// TIA Portal project "2022.06.13_步进电机定位指令" (V17)

(* hardware
DEVICE "S7-1200 station_1"  S7-1200 Station
   slot 0: "Rack_0"  S7-1200 Rack  Rack  V1.0
   slot 1: "PLC_1"  CPU 1212C DC/DC/DC  6ES7 212-1AE40-0XB0  V4.5
   slot 2: "AI 4x13BIT/AQ 2x14BIT_1"  SM 1234 AI4/AQ2  6ES7 234-4HE30-0XB0  V1.0
*)

// ===== PLC "PLC_1"  CPU 1212C DC/DC/DC =====

VAR_GLOBAL   // PLC tag table "默认变量表"
   "液位测量" AT %IW96 : Word;
   "百分比" AT %MD40 : DWord;
   "模拟量输出通道" AT %MD44 : UDInt;
   "所需频率(1)" AT %MD0 : Real;
   "压力2模拟输入通道" AT %IW100 : Int;
   "液位" AT %MD4 : Real;
   "频率" AT %MD8 : Real;
   "Tag_2" AT %MD12 : Real;
   "模拟量输出" AT %QW96 : Int;
   "设定液位值" AT %MD20 : Real;
   "实际液位值" AT %MD24 : Real;
   "轴_1_脉冲" AT %Q0.0 : Bool;
   "轴_1_方向" AT %Q0.1 : Bool;
   "轴_1_LowHwLimitSwitch" AT %I0.0 : Bool;
   "轴_1_HighHwLimitSwitch" AT %I0.1 : Bool;
   "轴_1_PassiveHomingSwitch" AT %I0.2 : Bool;
   "轴_1_归位开关" AT %I0.3 : Bool;
   "启用轴" AT %M0.0 : Bool;
   "完成位" AT %M0.1 : Bool;
   "Tag_1" AT %M0.2 : Bool;
   "回原点" AT %I1.0 : Bool;
   "Tag_3" AT %M0.4 : Bool;
   "Tag_4" AT %M0.5 : Bool;
   "Tag_5" AT %M0.3 : Bool;
   "触发绝对定位" AT %I1.1 : Bool;
   "Tag_7" AT %M0.6 : Bool;
   "指定位置" AT %MD30 : Real;
   "指定速度" AT %MD34 : Real;
   "Tag_6" AT %M0.7 : Bool;
   "Tag_8" AT %I1.2 : Bool;
   "Tag_9" AT %M1.0 : Bool;
   "触发相对位移指令" AT %I1.3 : Bool;
   "Tag_11" AT %M1.1 : Bool;
   "相对位置" AT %MD28 : Real;
   "速度" AT %MD32 : Real;
   "触发恒速" AT %I0.4 : Bool;
   "Tag_10" AT %M1.2 : Bool;
   "Tag_12" AT %MD36 : Real;
   "Tag_13" AT %I1.5 : Bool;
   "Tag_14" AT %M1.3 : Bool;
   "正点动" AT %I1.6 : Bool;
   "反点动" AT %I1.7 : Bool;
END_VAR

DATA_BLOCK "轴_1"   // DB2, Motion_DB
{ S7_Optimized_Access := 'TRUE' }
AUTHOR : SIMATIC
FAMILY : BasicMC
NAME : TO_PosAx
VERSION : 8.0
// stored: InstanceOfName TO_PositioningAxis
"TO_PositioningAxis"
BEGIN
END_DATA_BLOCK

ORGANIZATION_BLOCK "Main"   // OB1, LAD, ProgramCycle
TITLE = "Main Program Sweep (Cycle)"
{ S7_Optimized_Access := 'TRUE' }
VERSION : 0.1
   VAR_INPUT
      Initial_Call : Bool;   // Initial call of this OB
      Remanence : Bool;   // =True, if remanent data are available
   END_VAR
   VAR_TEMP   // added for the SCL form of the ladder/FBD networks
      _w1 : Bool;
   END_VAR
BEGIN

REGION Network 1
   // 启用轴，禁用轴,M0.0=1启用
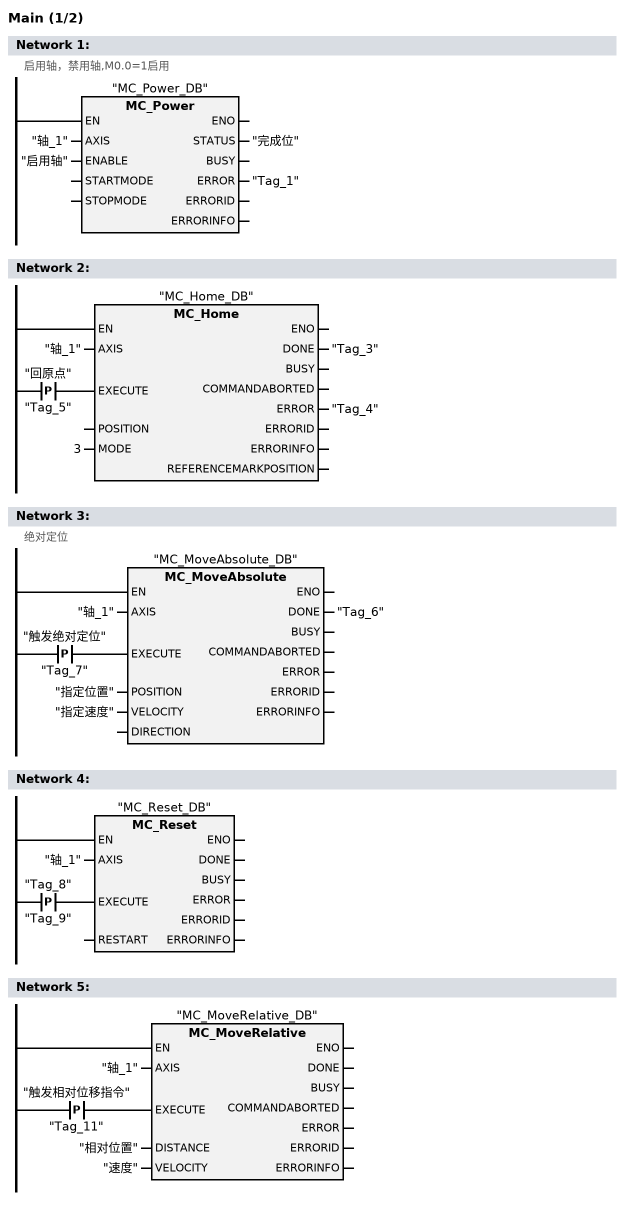
   "MC_Power_DB"(Axis := "轴_1", Enable := "启用轴", Status => "完成位", Error => "Tag_1");   // MC_Power
END_REGION

REGION Network 2
   #_w1 := "回原点" AND NOT "Tag_5";   // rising edge of "回原点"
   "Tag_5" := "回原点";
   "MC_Home_DB"(Axis := "轴_1", Execute := #_w1, Mode := 3, Done => "Tag_3", Error => "Tag_4");   // MC_Home
END_REGION

REGION Network 3
   // 绝对定位
   #_w1 := "触发绝对定位" AND NOT "Tag_7";   // rising edge of "触发绝对定位"
   "Tag_7" := "触发绝对定位";
   "MC_MoveAbsolute_DB"(Axis := "轴_1", Execute := #_w1, Position := "指定位置", Velocity := "指定速度", Done => "Tag_6");   // MC_MoveAbsolute
END_REGION

REGION Network 4
   #_w1 := "Tag_8" AND NOT "Tag_9";   // rising edge of "Tag_8"
   "Tag_9" := "Tag_8";
   "MC_Reset_DB"(Axis := "轴_1", Execute := #_w1);   // MC_Reset
END_REGION

REGION Network 5
   #_w1 := "触发相对位移指令" AND NOT "Tag_11";   // rising edge of "触发相对位移指令"
   "Tag_11" := "触发相对位移指令";
   "MC_MoveRelative_DB"(Axis := "轴_1", Execute := #_w1, Distance := "相对位置", Velocity := "速度");   // MC_MoveRelative
END_REGION

REGION Network 6
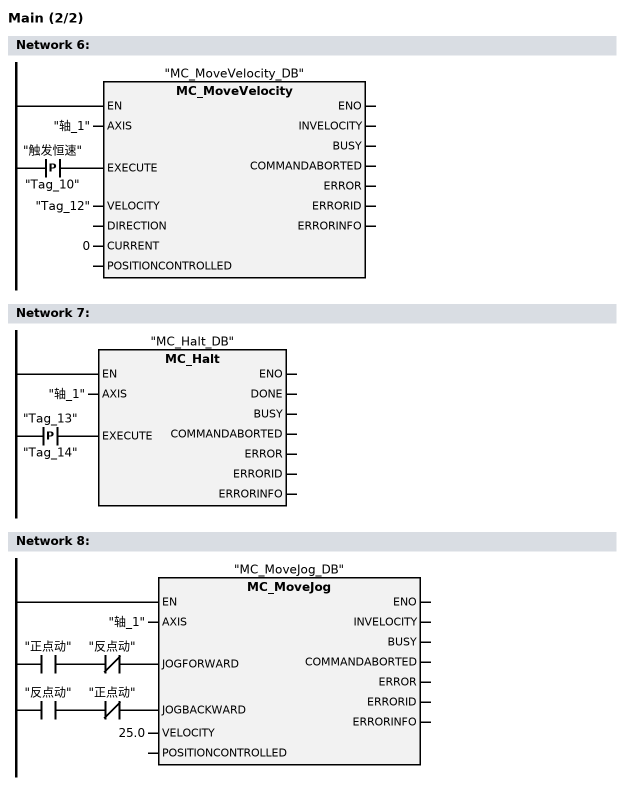
   #_w1 := "触发恒速" AND NOT "Tag_10";   // rising edge of "触发恒速"
   "Tag_10" := "触发恒速";
   "MC_MoveVelocity_DB"(Axis := "轴_1", Execute := #_w1, Velocity := "Tag_12", Current := 0);   // MC_MoveVelocity
END_REGION

REGION Network 7
   #_w1 := "Tag_13" AND NOT "Tag_14";   // rising edge of "Tag_13"
   "Tag_14" := "Tag_13";
   "MC_Halt_DB"(Axis := "轴_1", Execute := #_w1);   // MC_Halt
END_REGION

REGION Network 8
   "MC_MoveJog_DB"(Axis := "轴_1",   // MC_MoveJog
                   JogForward := "正点动" AND NOT "反点动",
                   JogBackward := "反点动" AND NOT "正点动",
                   Velocity := 25.0);
END_REGION
END_ORGANIZATION_BLOCK